Staubli VAL3: Entwicklungsmethodik.pjx

--- Entwicklungsmethodik.pjx ---
Parameters version=s8.3.1Cs9_BS885 stackSize=100000 millimeterUnit=true
Program file=pick.pgx
Program file=PickPlace.pgx
Program file=place.pgx
Program file=start.pgx
Program file=stop.pgx
Program file=TCPserver.pgx
Data file=Entwicklungsmethodik.dtx

--- Entwicklungsmethodik.dtx ---
mdesc mNomSpeed
frame fUserFrame = {x=701.757897, y=-321.609007, z=-207.673108, rx=-0.0947033, ry=0.52905, rz=90.111007, fatherId=world[0]}
tool tGreifer = {x=1.13686837721616E-13, y=-4.40536496171262E-13, z=110.500000000003, rx=-1.59027734073174E-14, ry=3.10104081442691E-14, rz=-2.14687465591809E-14, fatherId=flange[0], ioLink=ValveIO\valve1, ioOpen=0.05, ioClose=0.05}
pointRx pABPosition[12]
  [0] = {x=100, y=100, z=20, rx=180, rz=45, fatherId=fUserFrame[0]}
  [1] = {x=200, y=100, z=20, rx=180, rz=45, fatherId=fUserFrame[0]}
  [2] = {x=300, y=100, z=20, rx=180, rz=45, fatherId=fUserFrame[0]}
  [3] = {x=400, y=100, z=20, rx=180, rz=45, fatherId=fUserFrame[0]}
  [4] = {x=100, y=200, z=20, rx=180, rz=45, fatherId=fUserFrame[0]}
  [5] = {x=200, y=200, z=20, rx=180, rz=45, fatherId=fUserFrame[0]}
  [6] = {x=300, y=200, z=20, rx=180, rz=45, fatherId=fUserFrame[0]}
  [7] = {x=400, y=200, z=20, rx=180, rz=45, fatherId=fUserFrame[0]}
  [8] = {x=100, y=300, z=20, rx=180, rz=45, fatherId=fUserFrame[0]}
  [9] = {x=200, y=300, z=20, rx=180, rz=45, fatherId=fUserFrame[0]}
  [10] = {x=300, y=300, z=20, rx=180, rz=45, fatherId=fUserFrame[0]}
  [11] = {x=400, y=300, z=20, rx=180, rz=45, fatherId=fUserFrame[0]}
sio soTcpClient = {link=Socket\server0}
bool bNewData[2]
num nData[3]
bool bReady
jointRx jHome = {j3=90, j5=90}
mdesc mUsedSpeed
pointRx pPick = {z=20, rx=180, rz=45, fatherId=fUserFrame[0]}
trsf trApro = {z=-150}
pointRx pPlace = {z=20, rx=180, rz=45, fatherId=fUserFrame[0]}
bool bPick
num nX
num nY

--- start.pgx ---
program start()
begin

  clearBuffer(soTcpClient)
  movej(jHome,tGreifer,mUsedSpeed)

  taskCreate "TCP-Server", 10, TCPserver()

  taskCreate "p&p", 5, PickPlace()



  movej(jHome,tGreifer,mUsedSpeed)
  waitEndMove()

end

--- pick.pgx ---
program pick(num x_nX, num x_nY)
begin



  pPick.trsf.x = x_nX*100
  pPick.trsf.y = x_nY*100

  movej(appro(pPick,trApro),tGreifer, mUsedSpeed)
  movel(pPick, tGreifer, mUsedSpeed)
  close(tGreifer)
  movel(appro(pPick, trApro), tGreifer, mUsedSpeed)
  logMsg("Objekt aufgegriffen")





end

--- PickPlace.pgx ---
program PickPlace()
begin


  while true

    wait(bNewData)

    if bPick
      call pick(nX,nY)
    else
      call place(nX,nY)
    endIf


    bNewData = false
    bReady = true



  endWhile

end

--- place.pgx ---
program place(num x_nX, num x_nY)
begin



  pPlace.trsf.x = x_nX*100
  pPlace.trsf.y = x_nY*100

  movej(appro(pPlace,trApro),tGreifer, mUsedSpeed)
  movel(pPlace, tGreifer, mUsedSpeed)
  open(tGreifer)
  movel(appro(pPlace, trApro), tGreifer, mUsedSpeed)
  logMsg("Objekt abgelegt")





end

--- stop.pgx ---
program stop()
begin


end

--- TCPserver.pgx ---
program TCPserver()
  local num l_nStatus
  local num l_nBytesIn[24]
  local num l_nSuccBytes
begin
  // l_nBytesIn: 24 bit -> 3 byte
  // nData: 3
  while true
    logMsg("Schleife start")
    l_nStatus=sioGet(soTcpClient, l_nBytesIn)
    if l_nStatus>0
      // Write recieved bytes in data
      // Achtung bei mehr Bitlänge 24, 3 und globale Variable(nData) ändern
      logMsg("Empfangene Daten sind fehlerhaft",2)
      if(fromBinary(l_nBytesIn,24,"8.0l",nData)!=3)
      else
        logMsg("Daten über TCP/IP empfangen")
        // check if data is in limits
        // ...
        nX = limit(nData[0],1,4)
        nY = limit(nData[1],1,3)
        if nData[2]>0
          bPick = true
        else
          bPick = false
        endIf
        bReady = false
        bNewData = true
      endIf

      // tell client that robot is ready
      wait(bReady)

      //delay(2)
      l_nStatus=sioSet(soTcpClient, 1)
    endIf
  endWhile
end
